// TIA Portal V17 export
// export: Created 2024-08-26T21:07:19.6477514Z, ExportSetting WithDefaults, DisplayName Totally Integrated Automation Portal, DisplayVersion V17 Update 7, DisplayName TIA Portal Openness, DisplayVersion V17 Update 7, DisplayName TIA Portal Version Control Interface, DisplayVersion V17, DisplayName SINAMICS Startdrive Advanced, DisplayVersion V17 SP2, DisplayName SINAMICS Startdrive G110M, G120, G120C, G120D, G120P, G115D, DisplayVersion V17 SP2, DisplayName SINAMICS Startdrive G130, G150, S120, S150, SINAMICS MV, S210, DisplayVersion V17 SP2, DisplayName STEP 7 Professional, DisplayVersion V17 Update 7, DisplayName STEP 7 Safety, DisplayVersion V17 Update 6, DisplayName WinCC Advanced / Unified PC, DisplayVersion V17 Update 7
FUNCTION "MODIFY RECIPE" : Void   // FC6, LAD
{ S7_Optimized_Access := 'TRUE' }
VERSION : 0.1
// stored: AutoNumber true, IsIECCheckEnabled false, SetENOAutomatically false, UDAEnableTagReadback false
   VAR_TEMP   // added for the SCL form of the ladder/FBD networks
      _w1 : Bool;
      _w2 : Bool;
   END_VAR
BEGIN

REGION Network 1: ERASE A STEP
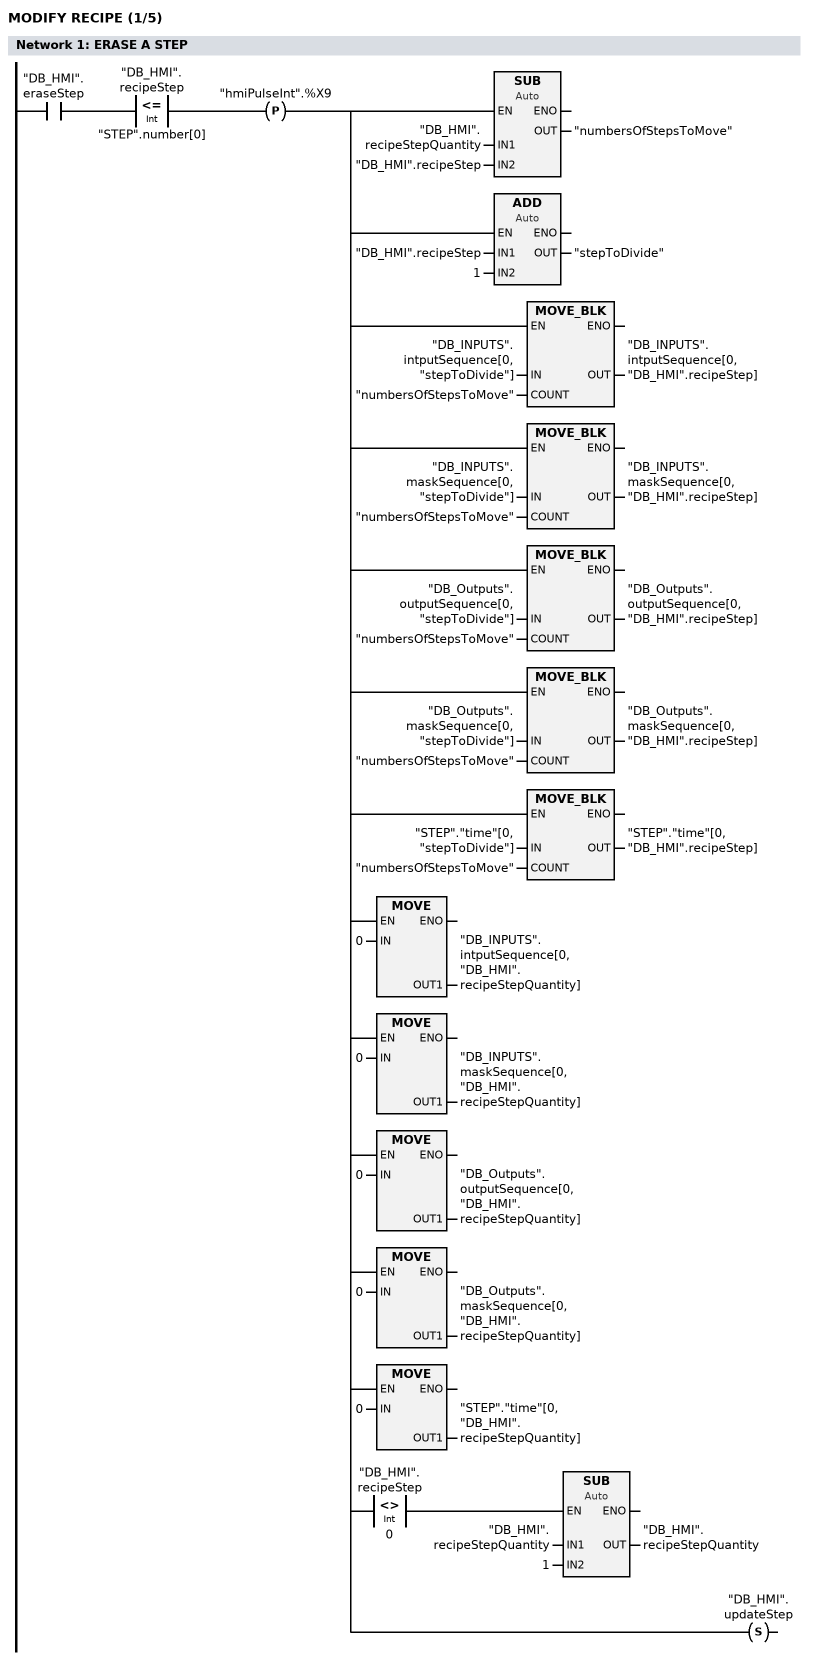
   #_w1 := "DB_HMI".eraseStep AND ("DB_HMI".recipeStep <= "STEP".number[0]);
   #_w2 := #_w1 AND NOT "hmiPulseInt".%X9;   // rising edge
   "hmiPulseInt".%X9 := #_w1;
   IF #_w2 THEN
       "numbersOfStepsToMove" := "DB_HMI".recipeStepQuantity - "DB_HMI".recipeStep;
       "stepToDivide" := "DB_HMI".recipeStep + 1;
       MOVE_BLK(IN := "DB_INPUTS".intputSequence[0, "stepToDivide"],
                COUNT := "numbersOfStepsToMove",
                OUT => "DB_INPUTS".intputSequence[0, "DB_HMI".recipeStep]);
       MOVE_BLK(IN := "DB_INPUTS".maskSequence[0, "stepToDivide"],
                COUNT := "numbersOfStepsToMove",
                OUT => "DB_INPUTS".maskSequence[0, "DB_HMI".recipeStep]);
       MOVE_BLK(IN := "DB_Outputs".outputSequence[0, "stepToDivide"],
                COUNT := "numbersOfStepsToMove",
                OUT => "DB_Outputs".outputSequence[0, "DB_HMI".recipeStep]);
       MOVE_BLK(IN := "DB_Outputs".maskSequence[0, "stepToDivide"],
                COUNT := "numbersOfStepsToMove",
                OUT => "DB_Outputs".maskSequence[0, "DB_HMI".recipeStep]);
       MOVE_BLK(IN := "STEP"."time"[0, "stepToDivide"],
                COUNT := "numbersOfStepsToMove",
                OUT => "STEP"."time"[0, "DB_HMI".recipeStep]);
       "DB_INPUTS".intputSequence[0, "DB_HMI".recipeStepQuantity] := 0;
       "DB_INPUTS".maskSequence[0, "DB_HMI".recipeStepQuantity] := 0;
       "DB_Outputs".outputSequence[0, "DB_HMI".recipeStepQuantity] := 0;
       "DB_Outputs".maskSequence[0, "DB_HMI".recipeStepQuantity] := 0;
       "STEP"."time"[0, "DB_HMI".recipeStepQuantity] := 0;
   END_IF;
   IF #_w2 AND ("DB_HMI".recipeStep <> 0) THEN
       "DB_HMI".recipeStepQuantity := "DB_HMI".recipeStepQuantity - 1;
   END_IF;
   IF #_w2 THEN "DB_HMI".updateStep := TRUE; END_IF;
END_REGION

REGION Network 2: ADD A STEP
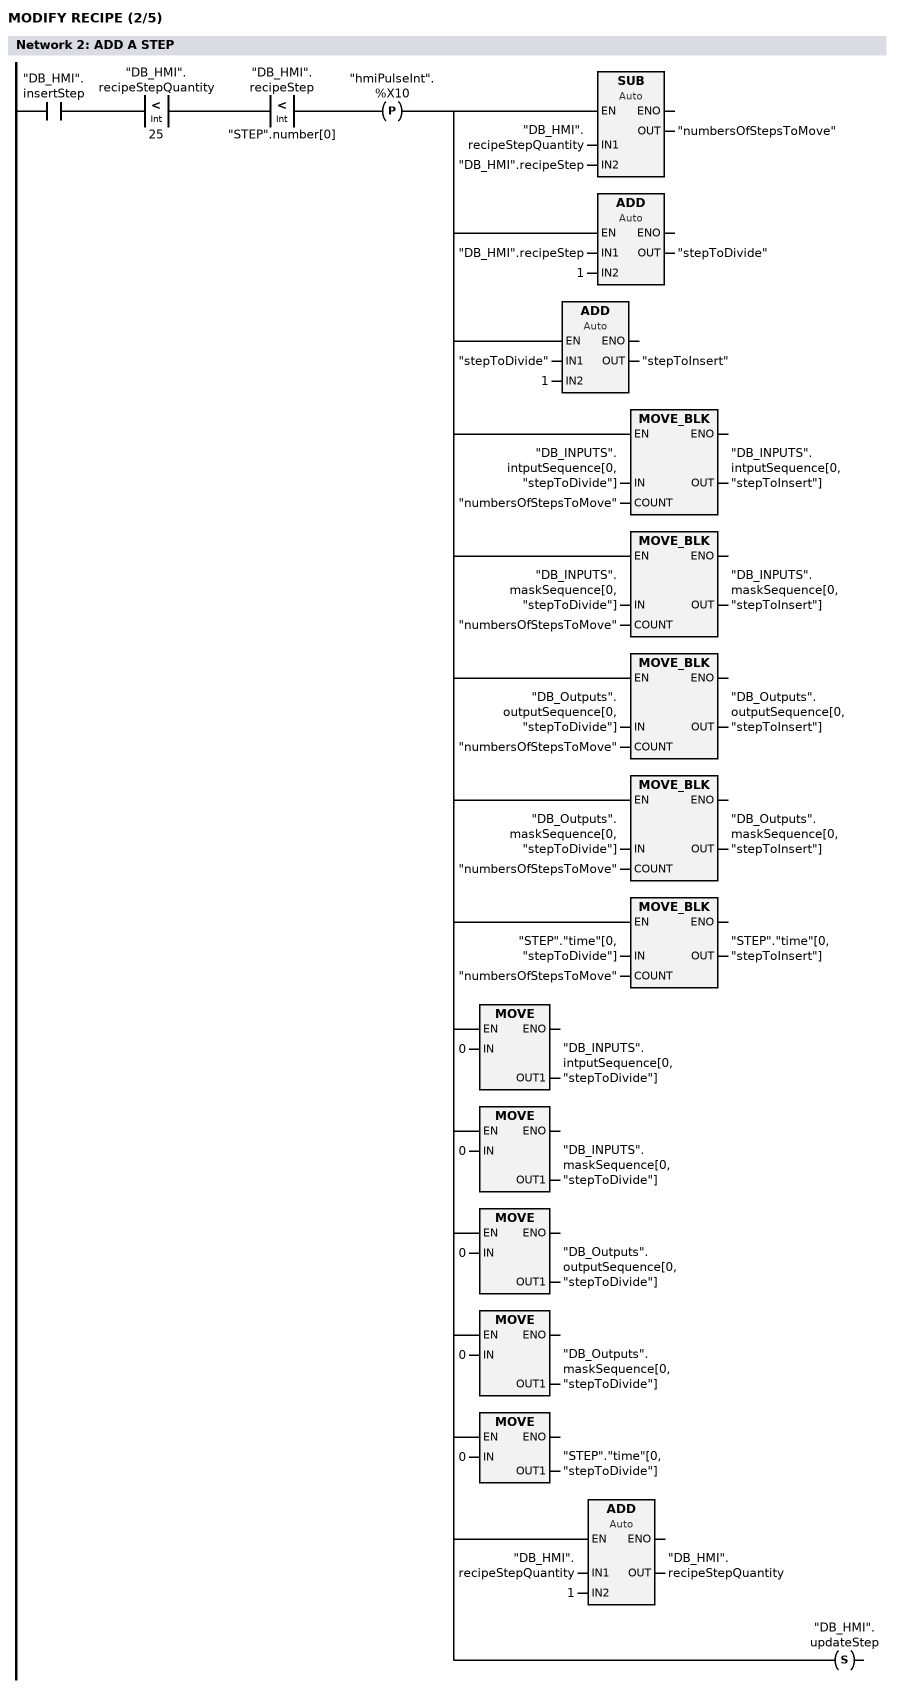
   #_w1 := "DB_HMI".insertStep AND ("DB_HMI".recipeStepQuantity < 25) AND ("DB_HMI".recipeStep < "STEP".number[0]);
   #_w2 := #_w1 AND NOT "hmiPulseInt".%X10;   // rising edge
   "hmiPulseInt".%X10 := #_w1;
   IF #_w2 THEN
       "numbersOfStepsToMove" := "DB_HMI".recipeStepQuantity - "DB_HMI".recipeStep;
       "stepToDivide" := "DB_HMI".recipeStep + 1;
       "stepToInsert" := "stepToDivide" + 1;
       MOVE_BLK(IN := "DB_INPUTS".intputSequence[0, "stepToDivide"],
                COUNT := "numbersOfStepsToMove",
                OUT => "DB_INPUTS".intputSequence[0, "stepToInsert"]);
       MOVE_BLK(IN := "DB_INPUTS".maskSequence[0, "stepToDivide"],
                COUNT := "numbersOfStepsToMove",
                OUT => "DB_INPUTS".maskSequence[0, "stepToInsert"]);
       MOVE_BLK(IN := "DB_Outputs".outputSequence[0, "stepToDivide"],
                COUNT := "numbersOfStepsToMove",
                OUT => "DB_Outputs".outputSequence[0, "stepToInsert"]);
       MOVE_BLK(IN := "DB_Outputs".maskSequence[0, "stepToDivide"],
                COUNT := "numbersOfStepsToMove",
                OUT => "DB_Outputs".maskSequence[0, "stepToInsert"]);
       MOVE_BLK(IN := "STEP"."time"[0, "stepToDivide"],
                COUNT := "numbersOfStepsToMove",
                OUT => "STEP"."time"[0, "stepToInsert"]);
       "DB_INPUTS".intputSequence[0, "stepToDivide"] := 0;
       "DB_INPUTS".maskSequence[0, "stepToDivide"] := 0;
       "DB_Outputs".outputSequence[0, "stepToDivide"] := 0;
       "DB_Outputs".maskSequence[0, "stepToDivide"] := 0;
       "STEP"."time"[0, "stepToDivide"] := 0;
       "DB_HMI".recipeStepQuantity := "DB_HMI".recipeStepQuantity + 1;
       "DB_HMI".updateStep := TRUE;
   END_IF;
END_REGION

REGION Network 3: COPY A STEP
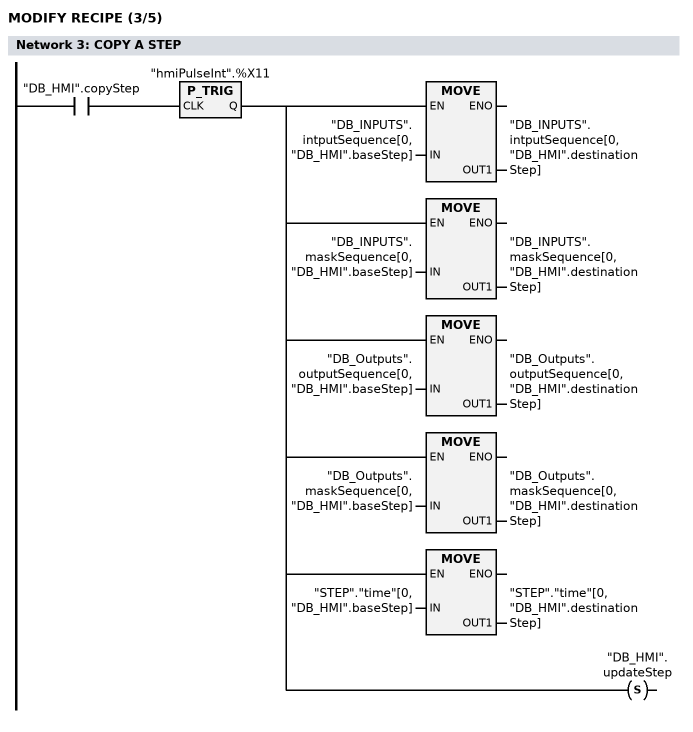
   RUNG wire#powerrail
      Contact( "DB_HMI".copyStep )
      P_Trig( "hmiPulseInt".%X11 )
      wire#w1
      Move(in := "DB_INPUTS".intputSequence[0, "DB_HMI".baseStep], out1 => "DB_INPUTS".intputSequence[0, "DB_HMI".destinationStep])
   END_RUNG
   RUNG wire#w1
      Move(in := "DB_INPUTS".maskSequence[0, "DB_HMI".baseStep], out1 => "DB_INPUTS".maskSequence[0, "DB_HMI".destinationStep])
   END_RUNG
   RUNG wire#w1
      Move(in := "DB_Outputs".outputSequence[0, "DB_HMI".baseStep], out1 => "DB_Outputs".outputSequence[0, "DB_HMI".destinationStep])
   END_RUNG
   RUNG wire#w1
      Move(in := "DB_Outputs".maskSequence[0, "DB_HMI".baseStep], out1 => "DB_Outputs".maskSequence[0, "DB_HMI".destinationStep])
   END_RUNG
   RUNG wire#w1
      Move(in := "STEP"."time"[0, "DB_HMI".baseStep], out1 => "STEP"."time"[0, "DB_HMI".destinationStep])
   END_RUNG
   RUNG wire#w1
      S_Coil( "DB_HMI".updateStep )
   END_RUNG
   // the same network as SCL:
   #_w1 := "DB_HMI".copyStep AND NOT "hmiPulseInt".%X11;   // rising edge
   "hmiPulseInt".%X11 := "DB_HMI".copyStep;
   IF #_w1 THEN
       "DB_INPUTS".intputSequence[0, "DB_HMI".destinationStep] := "DB_INPUTS".intputSequence[0, "DB_HMI".baseStep];
       "DB_INPUTS".maskSequence[0, "DB_HMI".destinationStep] := "DB_INPUTS".maskSequence[0, "DB_HMI".baseStep];
       "DB_Outputs".outputSequence[0, "DB_HMI".destinationStep] := "DB_Outputs".outputSequence[0, "DB_HMI".baseStep];
       "DB_Outputs".maskSequence[0, "DB_HMI".destinationStep] := "DB_Outputs".maskSequence[0, "DB_HMI".baseStep];
       "STEP"."time"[0, "DB_HMI".destinationStep] := "STEP"."time"[0, "DB_HMI".baseStep];
       "DB_HMI".updateStep := TRUE;
   END_IF;
END_REGION

REGION Network 4: COPY SEQUENCE (COPY PART NUMBER)
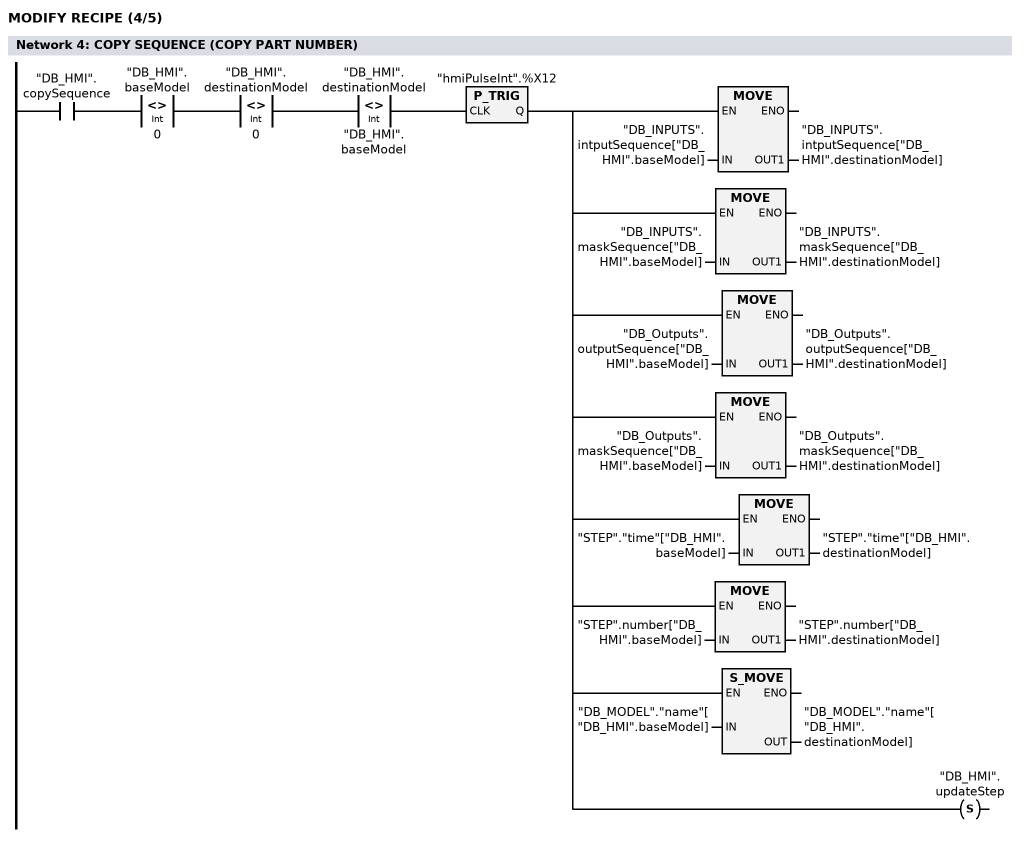
   RUNG wire#powerrail
      Contact( "DB_HMI".copySequence )
      { S7_Templates := "SrcType := Int" } NE_Contact(in1 := "DB_HMI".baseModel, in2 := 0)
      { S7_Templates := "SrcType := Int" } NE_Contact(in1 := "DB_HMI".destinationModel, in2 := 0)
      { S7_Templates := "SrcType := Int" } NE_Contact(in1 := "DB_HMI".destinationModel, in2 := "DB_HMI".baseModel)
      P_Trig( "hmiPulseInt".%X12 )
      wire#w1
      Move(in := "DB_INPUTS".intputSequence["DB_HMI".baseModel], out1 => "DB_INPUTS".intputSequence["DB_HMI".destinationModel])
   END_RUNG
   RUNG wire#w1
      Move(in := "DB_INPUTS".maskSequence["DB_HMI".baseModel], out1 => "DB_INPUTS".maskSequence["DB_HMI".destinationModel])
   END_RUNG
   RUNG wire#w1
      Move(in := "DB_Outputs".outputSequence["DB_HMI".baseModel], out1 => "DB_Outputs".outputSequence["DB_HMI".destinationModel])
   END_RUNG
   RUNG wire#w1
      Move(in := "DB_Outputs".maskSequence["DB_HMI".baseModel], out1 => "DB_Outputs".maskSequence["DB_HMI".destinationModel])
   END_RUNG
   RUNG wire#w1
      Move(in := "STEP"."time"["DB_HMI".baseModel], out1 => "STEP"."time"["DB_HMI".destinationModel])
   END_RUNG
   RUNG wire#w1
      Move(in := "STEP".number["DB_HMI".baseModel], out1 => "STEP".number["DB_HMI".destinationModel])
   END_RUNG
   RUNG wire#w1
      S_Move(in := "DB_MODEL"."name"["DB_HMI".baseModel], out => "DB_MODEL"."name"["DB_HMI".destinationModel])
   END_RUNG
   RUNG wire#w1
      S_Coil( "DB_HMI".updateStep )
   END_RUNG
   // the same network as SCL:
   #_w1 := "DB_HMI".copySequence AND ("DB_HMI".baseModel <> 0) AND ("DB_HMI".destinationModel <> 0) AND ("DB_HMI".destinationModel <> "DB_HMI".baseModel);
   #_w2 := #_w1 AND NOT "hmiPulseInt".%X12;   // rising edge
   "hmiPulseInt".%X12 := #_w1;
   IF #_w2 THEN
       "DB_INPUTS".intputSequence["DB_HMI".destinationModel] := "DB_INPUTS".intputSequence["DB_HMI".baseModel];
       "DB_INPUTS".maskSequence["DB_HMI".destinationModel] := "DB_INPUTS".maskSequence["DB_HMI".baseModel];
       "DB_Outputs".outputSequence["DB_HMI".destinationModel] := "DB_Outputs".outputSequence["DB_HMI".baseModel];
       "DB_Outputs".maskSequence["DB_HMI".destinationModel] := "DB_Outputs".maskSequence["DB_HMI".baseModel];
       "STEP"."time"["DB_HMI".destinationModel] := "STEP"."time"["DB_HMI".baseModel];
       "STEP".number["DB_HMI".destinationModel] := "STEP".number["DB_HMI".baseModel];
       "DB_MODEL"."name"["DB_HMI".destinationModel] := "DB_MODEL"."name"["DB_HMI".baseModel];
       "DB_HMI".updateStep := TRUE;
   END_IF;
END_REGION

REGION Network 5: COPY A STEP (#) FROM A PROGRAM (#) IN ANOTHER STEP (#) FROM ANOTHER PROGRAM (#)
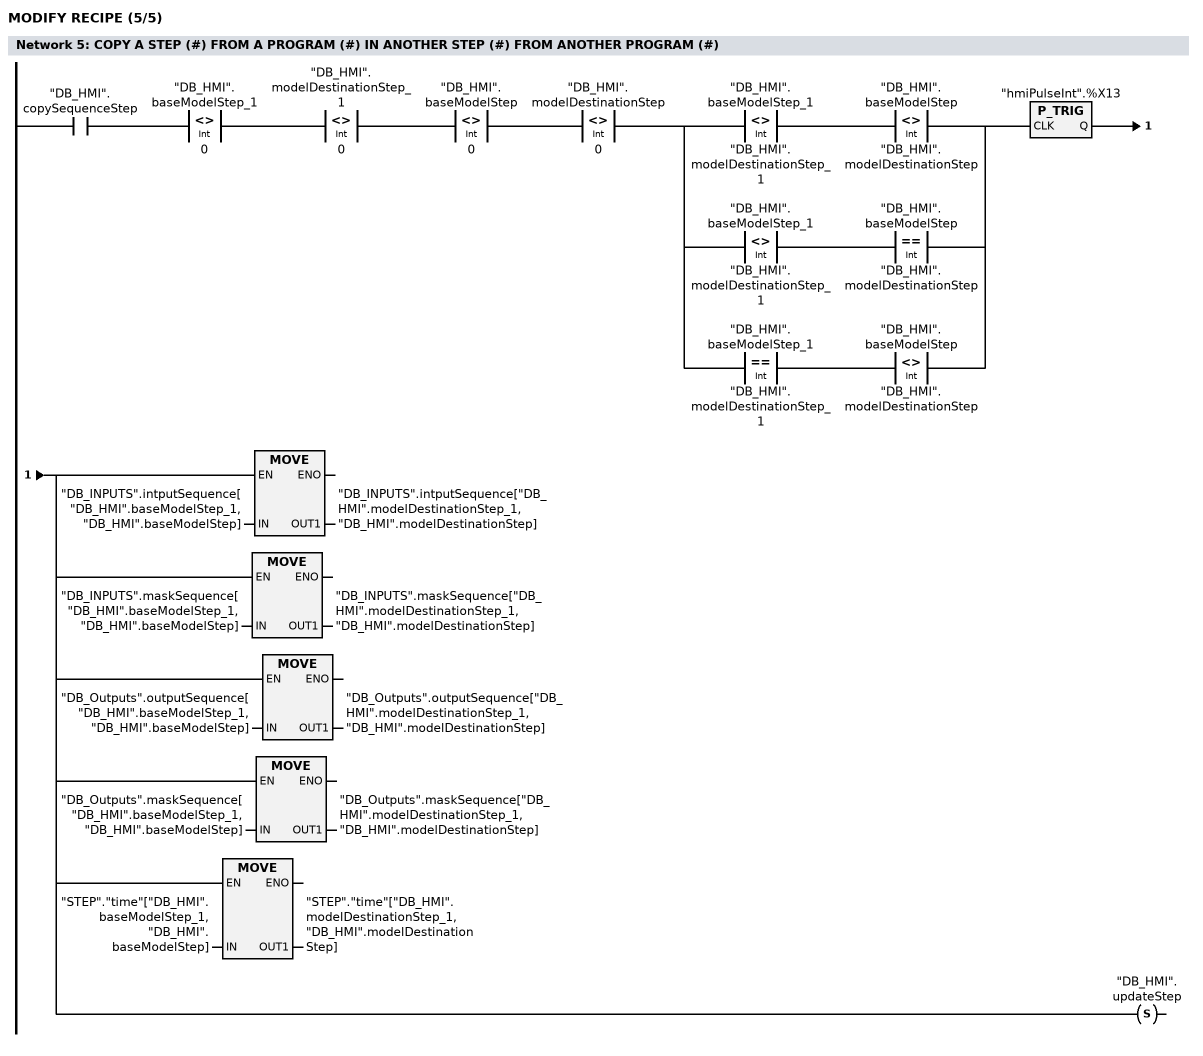
   RUNG wire#powerrail
      Contact( "DB_HMI".copySequenceStep )
      { S7_Templates := "SrcType := Int" } NE_Contact(in1 := "DB_HMI".baseModelStep_1, in2 := 0)
      { S7_Templates := "SrcType := Int" } NE_Contact(in1 := "DB_HMI".modelDestinationStep_1, in2 := 0)
      { S7_Templates := "SrcType := Int" } NE_Contact(in1 := "DB_HMI".baseModelStep, in2 := 0)
      { S7_Templates := "SrcType := Int" } NE_Contact(in1 := "DB_HMI".modelDestinationStep, in2 := 0)
      wire#w1
      { S7_Templates := "SrcType := Int" } NE_Contact(in1 := "DB_HMI".baseModelStep_1, in2 := "DB_HMI".modelDestinationStep_1)
      { S7_Templates := "SrcType := Int" } NE_Contact(in1 := "DB_HMI".baseModelStep, in2 := "DB_HMI".modelDestinationStep)
      wire#w2
      P_Trig( "hmiPulseInt".%X13 )
      wire#w3
      Move(in := "DB_INPUTS".intputSequence["DB_HMI".baseModelStep_1, "DB_HMI".baseModelStep], out1 => "DB_INPUTS".intputSequence["DB_HMI".modelDestinationStep_1, "DB_HMI".modelDestinationStep])
   END_RUNG
   RUNG wire#w1
      { S7_Templates := "SrcType := Int" } NE_Contact(in1 := "DB_HMI".baseModelStep_1, in2 := "DB_HMI".modelDestinationStep_1)
      { S7_Templates := "SrcType := Int" } EQ_Contact(in1 := "DB_HMI".baseModelStep, in2 := "DB_HMI".modelDestinationStep)
   END_RUNG wire#w2
   RUNG wire#w1
      { S7_Templates := "SrcType := Int" } EQ_Contact(in1 := "DB_HMI".baseModelStep_1, in2 := "DB_HMI".modelDestinationStep_1)
      { S7_Templates := "SrcType := Int" } NE_Contact(in1 := "DB_HMI".baseModelStep, in2 := "DB_HMI".modelDestinationStep)
   END_RUNG wire#w2
   RUNG wire#w3
      Move(in := "DB_INPUTS".maskSequence["DB_HMI".baseModelStep_1, "DB_HMI".baseModelStep], out1 => "DB_INPUTS".maskSequence["DB_HMI".modelDestinationStep_1, "DB_HMI".modelDestinationStep])
   END_RUNG
   RUNG wire#w3
      Move(in := "DB_Outputs".outputSequence["DB_HMI".baseModelStep_1, "DB_HMI".baseModelStep], out1 => "DB_Outputs".outputSequence["DB_HMI".modelDestinationStep_1, "DB_HMI".modelDestinationStep])
   END_RUNG
   RUNG wire#w3
      Move(in := "DB_Outputs".maskSequence["DB_HMI".baseModelStep_1, "DB_HMI".baseModelStep], out1 => "DB_Outputs".maskSequence["DB_HMI".modelDestinationStep_1, "DB_HMI".modelDestinationStep])
   END_RUNG
   RUNG wire#w3
      Move(in := "STEP"."time"["DB_HMI".baseModelStep_1, "DB_HMI".baseModelStep], out1 => "STEP"."time"["DB_HMI".modelDestinationStep_1, "DB_HMI".modelDestinationStep])
   END_RUNG
   RUNG wire#w3
      S_Coil( "DB_HMI".updateStep )
   END_RUNG
   // the same network as SCL:
   #_w1 := "DB_HMI".copySequenceStep AND ("DB_HMI".baseModelStep_1 <> 0) AND ("DB_HMI".modelDestinationStep_1 <> 0) AND ("DB_HMI".baseModelStep <> 0) AND ("DB_HMI".modelDestinationStep <> 0) AND ((("DB_HMI".baseModelStep_1 <> "DB_HMI".modelDestinationStep_1) AND ("DB_HMI".baseModelStep <> "DB_HMI".modelDestinationStep)) OR (("DB_HMI".baseModelStep_1 <> "DB_HMI".modelDestinationStep_1) AND ("DB_HMI".baseModelStep = "DB_HMI".modelDestinationStep)) OR (("DB_HMI".baseModelStep_1 = "DB_HMI".modelDestinationStep_1) AND ("DB_HMI".baseModelStep <> "DB_HMI".modelDestinationStep)));
   #_w2 := #_w1 AND NOT "hmiPulseInt".%X13;   // rising edge
   "hmiPulseInt".%X13 := #_w1;
   IF #_w2 THEN
       "DB_INPUTS".intputSequence["DB_HMI".modelDestinationStep_1, "DB_HMI".modelDestinationStep] := "DB_INPUTS".intputSequence["DB_HMI".baseModelStep_1, "DB_HMI".baseModelStep];
       "DB_INPUTS".maskSequence["DB_HMI".modelDestinationStep_1, "DB_HMI".modelDestinationStep] := "DB_INPUTS".maskSequence["DB_HMI".baseModelStep_1, "DB_HMI".baseModelStep];
       "DB_Outputs".outputSequence["DB_HMI".modelDestinationStep_1, "DB_HMI".modelDestinationStep] := "DB_Outputs".outputSequence["DB_HMI".baseModelStep_1, "DB_HMI".baseModelStep];
       "DB_Outputs".maskSequence["DB_HMI".modelDestinationStep_1, "DB_HMI".modelDestinationStep] := "DB_Outputs".maskSequence["DB_HMI".baseModelStep_1, "DB_HMI".baseModelStep];
       "STEP"."time"["DB_HMI".modelDestinationStep_1, "DB_HMI".modelDestinationStep] := "STEP"."time"["DB_HMI".baseModelStep_1, "DB_HMI".baseModelStep];
       "DB_HMI".updateStep := TRUE;
   END_IF;
END_REGION
END_FUNCTION
